TYPE ST_GCSingleProcessParam :
STRUCT
	LiftReady : ST_GCLiftPinAxisMoveAbsParam;
	SpinAlign : ST_GCSpinAxisMoveAbsParam;
	ProcessEntrySpin : ST_GCSpinAxisMoveAbsParam;
	ProcessEntryLift : ST_GCLiftPinAxisMoveAbsParam;
	SpinProcess : ST_GCSpinAxisMoveVelParam;
	ProcessExitLift : ST_GCLiftPinAxisMoveAbsParam;
	SpinStandby : ST_GCSpinAxisMoveAbsParam;
	SpinStopDeceleration : LREAL;
	LiftStopDeceleration : LREAL;
	StageTiming : ST_GCSingleProcessStageTimeConfigs;
	StopTimeout : TIME;
	ResetTimeout : TIME;
END_STRUCT
END_TYPE

(* stored: Version 1.1.0.1, ProductVersion 3.1.4026.18
   DUT ST_GCSingleProcessParam: Id {ce49dc48-904b-48bf-ae58-aca545aab98d} *)
